Yaskawa INFORM job: CLEANREQ.JBI

/JOB
//NAME CLEANREQ
///FOLDERNAME MASTER
//POS
///NPOS 3,0,0,0,0,0
///TOOL 4
///POSTYPE PULSE
///PULSE
C00000=-2,-80001,-25002,0,-113945,1
C00001=-119908,-80000,-25001,0,-113945,4
C00002=-119969,-12859,-35871,-1009,-70778,35
//INST
///DATE 2021/10/29 11:48
///ATTR SC,RO
///GROUP1 RB1
NOP
'Operator must clean the nozzle
MOVJ C00000 VJ=50.00
MOVJ C00001 VJ=50.00
MOVJ C00002 VJ=50.00
SET I010 0
END
